(* IEC 61131-3 sources: TSA-FMICS22/ahorn/test/benchmark/dissertation/augmentation/02/S, 2 files *)

(* ---- S.st ---- *)
PROGRAM SFEmergencyStop
VAR_INPUT
    Activate : BOOL;
    SEStopIn : BOOL;
    SStartReset : BOOL;
    SAutoReset : BOOL;
    Reset : BOOL;
END_VAR
VAR
    RTRIGatReset : RTRIG;
END_VAR
VAR_OUTPUT
    Ready : BOOL;
    SEStopOut : BOOL;
    Error : BOOL;
    DiagCode : WORD;
END_VAR
RTRIGatReset(CLK:=Reset);
IF NOT Activate THEN
    DiagCode := 16#0000;
ELSE
    CASE DiagCode OF
    16#0000:
        IF Activate THEN
            DiagCode := 16#8001;
        END_IF;
    16#8001:
        IF NOT SStartReset THEN
            DiagCode := 16#8002;
        ELSIF SStartReset AND NOT SEStopIn THEN
            DiagCode := 16#8004;
        ELSIF SEStopIn AND SStartReset THEN
            DiagCode := 16#8000;
        END_IF;
    16#8002:
        IF SEStopIn THEN
            DiagCode := 16#8003;
        END_IF;
    16#8003:
        IF Reset AND NOT RTRIGatReset.Q THEN
            DiagCode := 16#C001;
        ELSIF NOT SEStopIn THEN
            DiagCode := 16#8002;
        ELSIF RTRIGatReset.Q THEN
            DiagCode := change(16#8000, 16#8000);
        END_IF;
    16#C001:
        IF NOT Reset THEN
            DiagCode := 16#8003;
        END_IF;
    16#8004:
        IF SEStopIn AND NOT SAutoReset THEN
            DiagCode := 16#8005;
        ELSIF SEStopIn AND SAutoReset THEN
            DiagCode := 16#8000;
        END_IF;
    16#8005:
        IF Reset AND NOT RTRIGatReset.Q THEN
            DiagCode := 16#C002;
        ELSIF NOT SEStopIn THEN
            DiagCode := 16#8004;
        ELSIF RTRIGatReset.Q OR SAutoReset THEN
            DiagCode := 16#8000;
        END_IF;
    16#C002:
        IF NOT Reset THEN
            DiagCode := 16#8005;
        END_IF;
    16#8000:
        IF NOT SEStopIn THEN
            DiagCode := 16#8004;
        END_IF;
    END_CASE;
END_IF;
CASE DiagCode OF
16#0000:
    Ready := FALSE;
    Error := FALSE;
    SEStopOut := FALSE;
16#8001:
    Ready := TRUE;
    Error := FALSE;
    SEStopOut := FALSE;
16#8002:
    Ready := TRUE;
    Error := FALSE;
    SEStopOut := FALSE;
16#8003:
    Ready := TRUE;
    Error := FALSE;
    SEStopOut := FALSE;
16#C001:
    Ready := TRUE;
    Error := TRUE;
    SEStopOut := FALSE;
16#8004:
    Ready := TRUE;
    Error := FALSE;
    SEStopOut := FALSE;
16#8005:
    Ready := TRUE;
    Error := FALSE;
    SEStopOut := FALSE;
16#C002:
    Ready := TRUE;
    Error := TRUE;
    SEStopOut := FALSE;
16#8000:
    Ready := TRUE;
    Error := FALSE;
    SEStopOut := TRUE;
END_CASE;
END_PROGRAM

FUNCTION_BLOCK RTRIG
VAR_INPUT
    CLK : BOOL;
END_VAR
VAR
    M : BOOL;
END_VAR
VAR_OUTPUT
    Q : BOOL;
END_VAR
    Q := CLK AND NOT M;
    M := CLK;
END_FUNCTION_BLOCK

(* ---- S2.st ---- *)
PROGRAM SFEmergencyStop
VAR_INPUT
    Activate : BOOL;
    SEStopIn : BOOL;
    SStartReset : BOOL;
    SAutoReset : BOOL;
    Reset : BOOL;
END_VAR
VAR
    RTRIGatReset : RTRIG;
END_VAR
VAR_OUTPUT
    Ready : BOOL;
    SEStopOut : BOOL;
    Error : BOOL;
    DiagCode : WORD;
END_VAR
RTRIGatReset(CLK:=Reset);
IF change(NOT Activate, FALSE) THEN
    DiagCode := 16#0000;
ELSE
    CASE DiagCode OF
    16#0000:
        IF change(Activate, TRUE) THEN
            DiagCode := 16#8001;
        END_IF;
    16#8001:
        IF NOT SStartReset THEN
            DiagCode := 16#8002;
        ELSIF SStartReset AND NOT SEStopIn THEN
            DiagCode := 16#8004;
        ELSIF SEStopIn AND SStartReset THEN
            DiagCode := 16#8000;
        END_IF;
    16#8002:
        IF SEStopIn THEN
            DiagCode := 16#8003;
        END_IF;
    16#8003:
        IF Reset AND NOT RTRIGatReset.Q THEN
            DiagCode := 16#C001;
        ELSIF NOT SEStopIn THEN
            DiagCode := 16#8002;
        ELSIF RTRIGatReset.Q THEN
            DiagCode := change(16#8000, 16#8000);
        END_IF;
    16#C001:
        IF NOT Reset THEN
            DiagCode := 16#8003;
        END_IF;
    16#8004:
        IF SEStopIn AND NOT SAutoReset THEN
            DiagCode := 16#8005;
        ELSIF SEStopIn AND SAutoReset THEN
            DiagCode := 16#8000;
        END_IF;
    16#8005:
        IF Reset AND NOT RTRIGatReset.Q THEN
            DiagCode := 16#C002;
        ELSIF NOT SEStopIn THEN
            DiagCode := 16#8004;
        ELSIF RTRIGatReset.Q OR SAutoReset THEN
            DiagCode := 16#8000;
        END_IF;
    16#C002:
        IF NOT Reset THEN
            DiagCode := 16#8005;
        END_IF;
    16#8000:
        IF NOT SEStopIn THEN
            DiagCode := 16#8004;
        END_IF;
    END_CASE;
END_IF;
CASE DiagCode OF
16#0000:
    Ready := FALSE;
    Error := FALSE;
    SEStopOut := FALSE;
16#8001:
    Ready := TRUE;
    Error := FALSE;
    SEStopOut := FALSE;
16#8002:
    Ready := TRUE;
    Error := FALSE;
    SEStopOut := FALSE;
16#8003:
    Ready := TRUE;
    Error := FALSE;
    SEStopOut := FALSE;
16#C001:
    Ready := TRUE;
    Error := TRUE;
    SEStopOut := FALSE;
16#8004:
    Ready := TRUE;
    Error := FALSE;
    SEStopOut := FALSE;
16#8005:
    Ready := TRUE;
    Error := FALSE;
    SEStopOut := FALSE;
16#C002:
    Ready := TRUE;
    Error := TRUE;
    SEStopOut := FALSE;
16#8000:
    Ready := TRUE;
    Error := FALSE;
    SEStopOut := TRUE;
END_CASE;
END_PROGRAM

FUNCTION_BLOCK RTRIG
VAR_INPUT
    CLK : BOOL;
END_VAR
VAR
    M : BOOL;
END_VAR
VAR_OUTPUT
    Q : BOOL;
END_VAR
    Q := CLK AND NOT M;
    M := CLK;
END_FUNCTION_BLOCK
